INTERFACE I_ServerConfig EXTENDS I_SessionMiddlewareConfig, I_ServerResponseConfig, I_RpcMiddlewareConfig, I_RpcResponseManagerConfig, I_PendingResponseManagerConfig, I_ChunkedResponseManagerConfig, I_ChunkedRequestsManagerConfig

END_INTERFACE

(* stored: Version 1.1.0.1, ProductVersion 3.1.4024.12
   Itf I_ServerConfig: Id {39c7717a-a112-4a65-95ac-09aab042aac6} *)
